// TIA Portal V17 export
// export: Created 2024-08-29T18:23:43.7048748Z, ExportSetting WithDefaults, DisplayName Totally Integrated Automation Portal, DisplayVersion V17 Update 7, DisplayName TIA Portal Openness, DisplayVersion V17 Update 7, DisplayName TIA Portal Version Control Interface, DisplayVersion V17, DisplayName SINAMICS Startdrive Advanced, DisplayVersion V17 SP2, DisplayName SINAMICS Startdrive G110M, G120, G120C, G120D, G120P, G115D, DisplayVersion V17 SP2, DisplayName SINAMICS Startdrive G130, G150, S120, S150, SINAMICS MV, S210, DisplayVersion V17 SP2, DisplayName STEP 7 Professional, DisplayVersion V17 Update 7, DisplayName STEP 7 Safety, DisplayVersion V17 Update 6, DisplayName WinCC Advanced / Unified PC, DisplayVersion V17 Update 7
FUNCTION "analogSignals" : Void   // FC16, LAD
{ S7_Optimized_Access := 'TRUE' }
VERSION : 0.1
// stored: AutoNumber true, IsIECCheckEnabled false, SetENOAutomatically false, UDAEnableTagReadback false
   VAR_TEMP
      minimumScaleRangeArray : Array[0..9] of Real;
      maximumScaleRangeArray : Array[0..9] of Real;
      i : Int;
   END_VAR
BEGIN

REGION Network 1 (SCL): Initialize Temp Values
   FOR #i := 0 TO 9 DO
       #minimumScaleRangeArray[#i] := 0;
       #maximumScaleRangeArray[#i] := 0;
   END_FOR;
END_REGION

REGION Network 2: Load Cell Adquisition
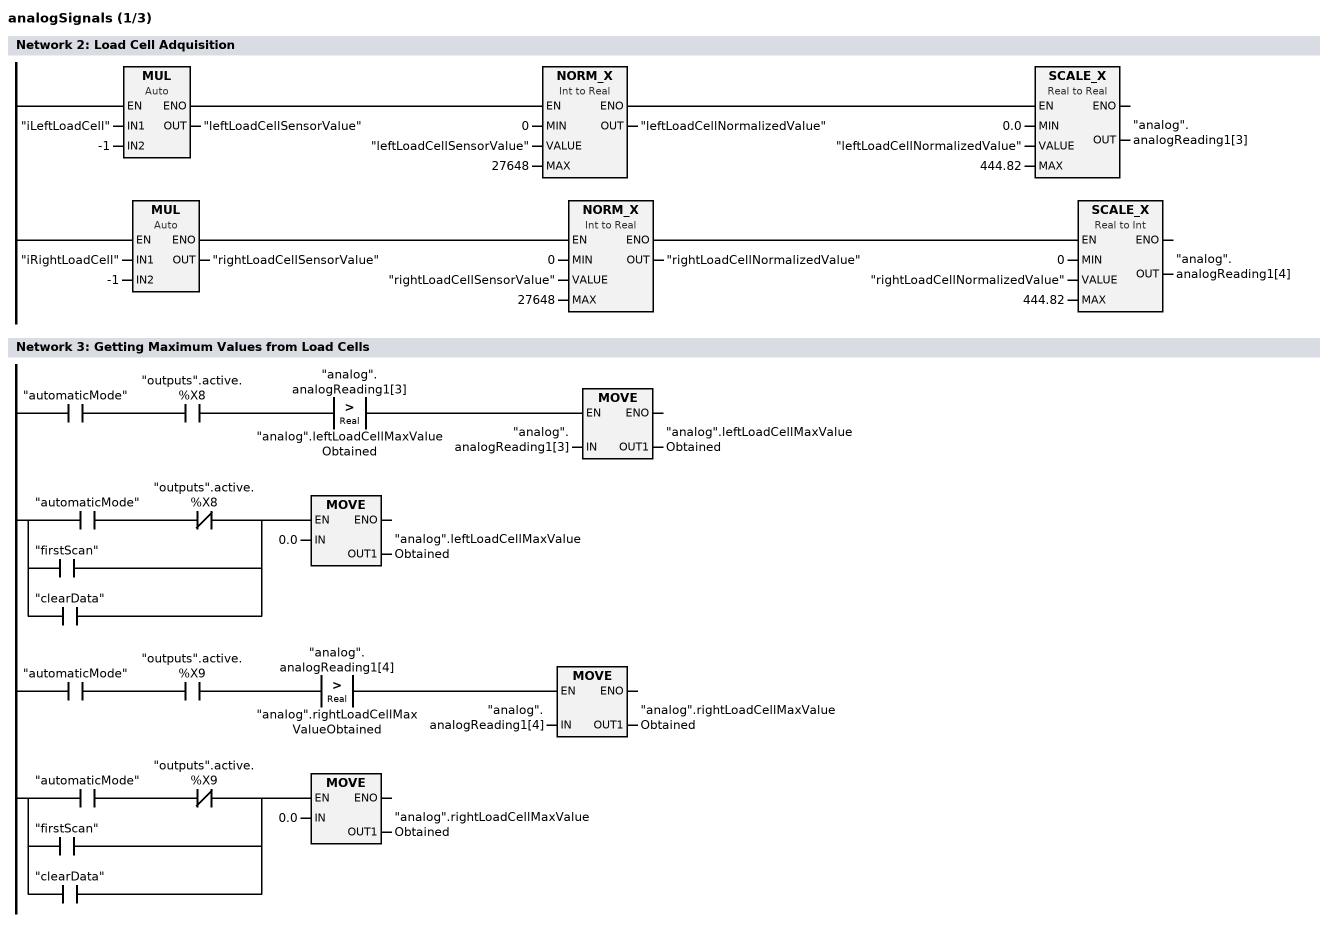
   RUNG wire#powerrail
      Mul(in1 := "iLeftLoadCell", in2 := -1, out => "leftLoadCellSensorValue")
      { S7_Templates := "[SrcType := Int, DestType := Real]" } Normalize(min := 0, value := "leftLoadCellSensorValue", max := 27648, out => "leftLoadCellNormalizedValue")
      { S7_Templates := "[SrcType := Real, DestType := Real]" } Scale(min := 0.0, value := "leftLoadCellNormalizedValue", max := 444.82, out => "analog".analogReading1[3])
   END_RUNG
   RUNG wire#powerrail
      Mul(in1 := "iRightLoadCell", in2 := -1, out => "rightLoadCellSensorValue")
      { S7_Templates := "[SrcType := Int, DestType := Real]" } Normalize(min := 0, value := "rightLoadCellSensorValue", max := 27648, out => "rightLoadCellNormalizedValue")
      { S7_Templates := "[SrcType := Real, DestType := Int]" } Scale(min := 0, value := "rightLoadCellNormalizedValue", max := 444.82, out => "analog".analogReading1[4])
   END_RUNG
   // the same network as SCL:
   "leftLoadCellSensorValue" := "iLeftLoadCell" * (-1);
   "leftLoadCellNormalizedValue" := NORM_X(MIN := 0, VALUE := "leftLoadCellSensorValue", MAX := 27648);
   "analog".analogReading1[3] := SCALE_X(MIN := 0.0, VALUE := "leftLoadCellNormalizedValue", MAX := 444.82);
   "rightLoadCellSensorValue" := "iRightLoadCell" * (-1);
   "rightLoadCellNormalizedValue" := NORM_X(MIN := 0, VALUE := "rightLoadCellSensorValue", MAX := 27648);
   "analog".analogReading1[4] := SCALE_X(MIN := 0, VALUE := "rightLoadCellNormalizedValue", MAX := 444.82);
END_REGION

REGION Network 3: Getting Maximum Values from Load Cells
   RUNG wire#powerrail
      Contact( "automaticMode" )
      Contact( "outputs".active.%X8 )
      { S7_Templates := "SrcType := Real" } GT_Contact(in1 := "analog".analogReading1[3], in2 := "analog".leftLoadCellMaxValueObtained)
      Move(in := "analog".analogReading1[3], out1 => "analog".leftLoadCellMaxValueObtained)
   END_RUNG
   RUNG wire#powerrail
      Contact( "automaticMode" )
      I_Contact( "outputs".active.%X8 )
      wire#w1
      Move(in := 0.0, out1 => "analog".leftLoadCellMaxValueObtained)
   END_RUNG
   RUNG wire#powerrail
      Contact( "firstScan" )
   END_RUNG wire#w1
   RUNG wire#powerrail
      Contact( "clearData" )
   END_RUNG wire#w1
   RUNG wire#powerrail
      Contact( "automaticMode" )
      Contact( "outputs".active.%X9 )
      { S7_Templates := "SrcType := Real" } GT_Contact(in1 := "analog".analogReading1[4], in2 := "analog".rightLoadCellMaxValueObtained)
      Move(in := "analog".analogReading1[4], out1 => "analog".rightLoadCellMaxValueObtained)
   END_RUNG
   RUNG wire#powerrail
      Contact( "automaticMode" )
      I_Contact( "outputs".active.%X9 )
      wire#w2
      Move(in := 0.0, out1 => "analog".rightLoadCellMaxValueObtained)
   END_RUNG
   RUNG wire#powerrail
      Contact( "firstScan" )
   END_RUNG wire#w2
   RUNG wire#powerrail
      Contact( "clearData" )
   END_RUNG wire#w2
   // the same network as SCL:
   IF "automaticMode" AND "outputs".active.%X8 AND ("analog".analogReading1[3] > "analog".leftLoadCellMaxValueObtained) THEN
       "analog".leftLoadCellMaxValueObtained := "analog".analogReading1[3];
   END_IF;
   IF ("automaticMode" AND NOT "outputs".active.%X8) OR "firstScan" OR "clearData" THEN
       "analog".leftLoadCellMaxValueObtained := 0.0;
   END_IF;
   IF "automaticMode" AND "outputs".active.%X9 AND ("analog".analogReading1[4] > "analog".rightLoadCellMaxValueObtained) THEN
       "analog".rightLoadCellMaxValueObtained := "analog".analogReading1[4];
   END_IF;
   IF ("automaticMode" AND NOT "outputs".active.%X9) OR "firstScan" OR "clearData" THEN
       "analog".rightLoadCellMaxValueObtained := 0.0;
   END_IF;
END_REGION

REGION Network 4: Effort OK/NOK Evaluation
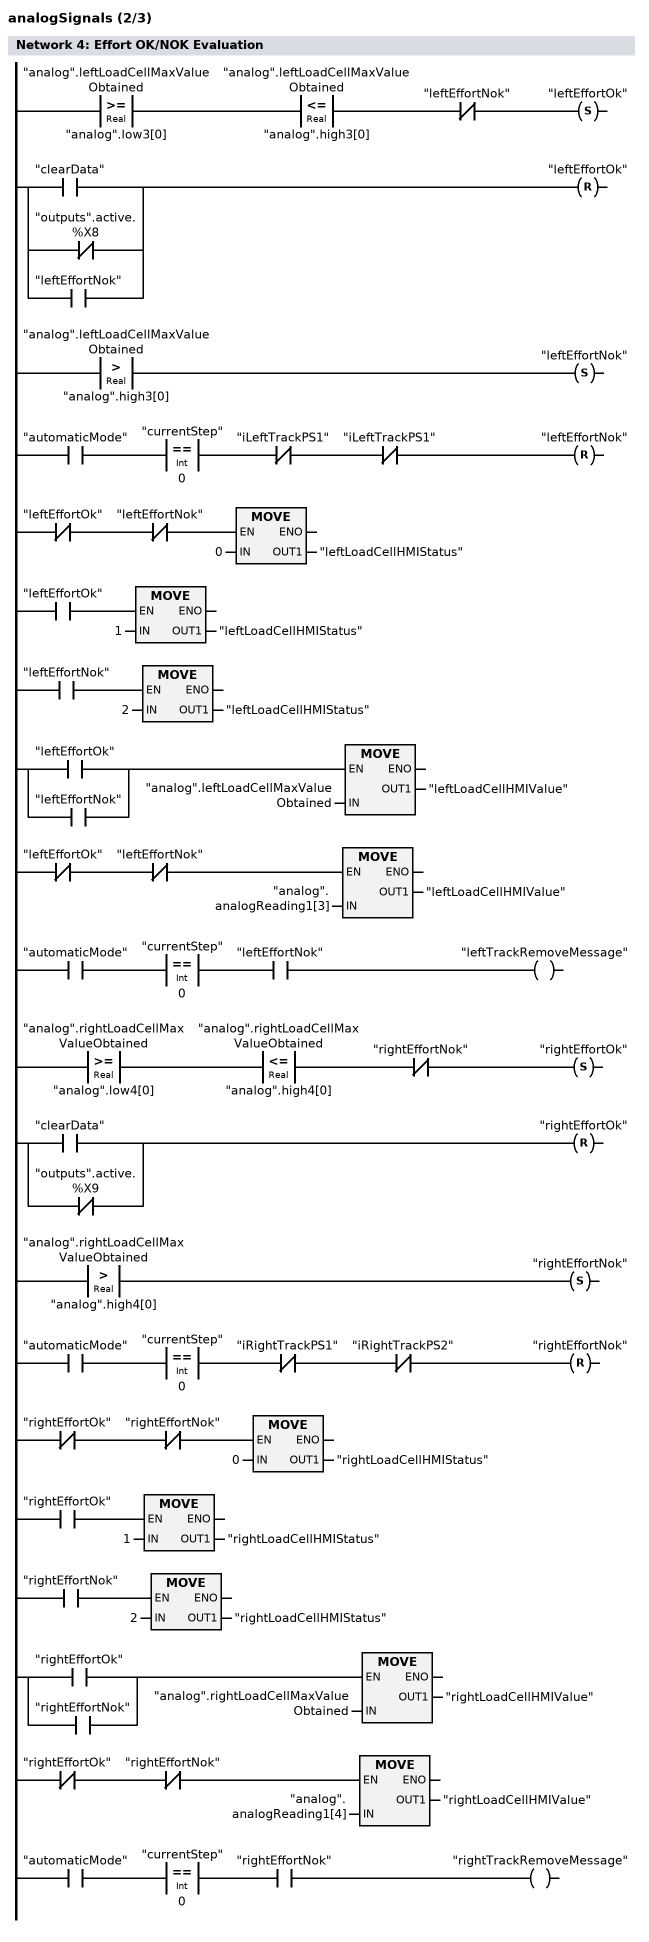
   RUNG wire#powerrail
      { S7_Templates := "SrcType := Real" } GE_Contact(in1 := "analog".leftLoadCellMaxValueObtained, in2 := "analog".low3[0])
      { S7_Templates := "SrcType := Real" } LE_Contact(in1 := "analog".leftLoadCellMaxValueObtained, in2 := "analog".high3[0])
      I_Contact( "leftEffortNok" )
      S_Coil( "leftEffortOk" )
   END_RUNG
   RUNG wire#powerrail
      Contact( "clearData" )
      wire#w1
      R_Coil( "leftEffortOk" )
   END_RUNG
   RUNG wire#powerrail
      I_Contact( "outputs".active.%X8 )
   END_RUNG wire#w1
   RUNG wire#powerrail
      Contact( "leftEffortNok" )
   END_RUNG wire#w1
   RUNG wire#powerrail
      { S7_Templates := "SrcType := Real" } GT_Contact(in1 := "analog".leftLoadCellMaxValueObtained, in2 := "analog".high3[0])
      S_Coil( "leftEffortNok" )
   END_RUNG
   RUNG wire#powerrail
      Contact( "automaticMode" )
      { S7_Templates := "SrcType := Int" } EQ_Contact(in1 := "currentStep", in2 := 0)
      I_Contact( "iLeftTrackPS1" )
      I_Contact( "iLeftTrackPS1" )
      R_Coil( "leftEffortNok" )
   END_RUNG
   RUNG wire#powerrail
      I_Contact( "leftEffortOk" )
      I_Contact( "leftEffortNok" )
      Move(in := 0, out1 => "leftLoadCellHMIStatus")
   END_RUNG
   RUNG wire#powerrail
      Contact( "leftEffortOk" )
      Move(in := 1, out1 => "leftLoadCellHMIStatus")
   END_RUNG
   RUNG wire#powerrail
      Contact( "leftEffortNok" )
      Move(in := 2, out1 => "leftLoadCellHMIStatus")
   END_RUNG
   RUNG wire#powerrail
      Contact( "leftEffortOk" )
      wire#w2
      Move(in := "analog".leftLoadCellMaxValueObtained, out1 => "leftLoadCellHMIValue")
   END_RUNG
   RUNG wire#powerrail
      Contact( "leftEffortNok" )
   END_RUNG wire#w2
   RUNG wire#powerrail
      I_Contact( "leftEffortOk" )
      I_Contact( "leftEffortNok" )
      Move(in := "analog".analogReading1[3], out1 => "leftLoadCellHMIValue")
   END_RUNG
   RUNG wire#powerrail
      Contact( "automaticMode" )
      { S7_Templates := "SrcType := Int" } EQ_Contact(in1 := "currentStep", in2 := 0)
      Contact( "leftEffortNok" )
      Coil( "leftTrackRemoveMessage" )
   END_RUNG
   RUNG wire#powerrail
      { S7_Templates := "SrcType := Real" } GE_Contact(in1 := "analog".rightLoadCellMaxValueObtained, in2 := "analog".low4[0])
      { S7_Templates := "SrcType := Real" } LE_Contact(in1 := "analog".rightLoadCellMaxValueObtained, in2 := "analog".high4[0])
      I_Contact( "rightEffortNok" )
      S_Coil( "rightEffortOk" )
   END_RUNG
   RUNG wire#powerrail
      Contact( "clearData" )
      wire#w3
      R_Coil( "rightEffortOk" )
   END_RUNG
   RUNG wire#powerrail
      I_Contact( "outputs".active.%X9 )
   END_RUNG wire#w3
   RUNG wire#powerrail
      { S7_Templates := "SrcType := Real" } GT_Contact(in1 := "analog".rightLoadCellMaxValueObtained, in2 := "analog".high4[0])
      S_Coil( "rightEffortNok" )
   END_RUNG
   RUNG wire#powerrail
      Contact( "automaticMode" )
      { S7_Templates := "SrcType := Int" } EQ_Contact(in1 := "currentStep", in2 := 0)
      I_Contact( "iRightTrackPS1" )
      I_Contact( "iRightTrackPS2" )
      R_Coil( "rightEffortNok" )
   END_RUNG
   RUNG wire#powerrail
      I_Contact( "rightEffortOk" )
      I_Contact( "rightEffortNok" )
      Move(in := 0, out1 => "rightLoadCellHMIStatus")
   END_RUNG
   RUNG wire#powerrail
      Contact( "rightEffortOk" )
      Move(in := 1, out1 => "rightLoadCellHMIStatus")
   END_RUNG
   RUNG wire#powerrail
      Contact( "rightEffortNok" )
      Move(in := 2, out1 => "rightLoadCellHMIStatus")
   END_RUNG
   RUNG wire#powerrail
      Contact( "rightEffortOk" )
      wire#w4
      Move(in := "analog".rightLoadCellMaxValueObtained, out1 => "rightLoadCellHMIValue")
   END_RUNG
   RUNG wire#powerrail
      Contact( "rightEffortNok" )
   END_RUNG wire#w4
   RUNG wire#powerrail
      I_Contact( "rightEffortOk" )
      I_Contact( "rightEffortNok" )
      Move(in := "analog".analogReading1[4], out1 => "rightLoadCellHMIValue")
   END_RUNG
   RUNG wire#powerrail
      Contact( "automaticMode" )
      { S7_Templates := "SrcType := Int" } EQ_Contact(in1 := "currentStep", in2 := 0)
      Contact( "rightEffortNok" )
      Coil( "rightTrackRemoveMessage" )
   END_RUNG
   // the same network as SCL:
   IF ("analog".leftLoadCellMaxValueObtained >= "analog".low3[0]) AND ("analog".leftLoadCellMaxValueObtained <= "analog".high3[0]) AND NOT "leftEffortNok" THEN
       "leftEffortOk" := TRUE;
   END_IF;
   IF "clearData" OR NOT "outputs".active.%X8 OR "leftEffortNok" THEN "leftEffortOk" := FALSE; END_IF;
   IF "analog".leftLoadCellMaxValueObtained > "analog".high3[0] THEN "leftEffortNok" := TRUE; END_IF;
   IF "automaticMode" AND ("currentStep" = 0) AND NOT "iLeftTrackPS1" AND NOT "iLeftTrackPS1" THEN
       "leftEffortNok" := FALSE;
   END_IF;
   IF NOT "leftEffortOk" AND NOT "leftEffortNok" THEN "leftLoadCellHMIStatus" := 0; END_IF;
   IF "leftEffortOk" THEN "leftLoadCellHMIStatus" := 1; END_IF;
   IF "leftEffortNok" THEN "leftLoadCellHMIStatus" := 2; END_IF;
   IF "leftEffortOk" OR "leftEffortNok" THEN
       "leftLoadCellHMIValue" := "analog".leftLoadCellMaxValueObtained;
   END_IF;
   IF NOT "leftEffortOk" AND NOT "leftEffortNok" THEN
       "leftLoadCellHMIValue" := "analog".analogReading1[3];
   END_IF;
   "leftTrackRemoveMessage" := "automaticMode" AND ("currentStep" = 0) AND "leftEffortNok";
   IF ("analog".rightLoadCellMaxValueObtained >= "analog".low4[0]) AND ("analog".rightLoadCellMaxValueObtained <= "analog".high4[0]) AND NOT "rightEffortNok" THEN
       "rightEffortOk" := TRUE;
   END_IF;
   IF "clearData" OR NOT "outputs".active.%X9 THEN "rightEffortOk" := FALSE; END_IF;
   IF "analog".rightLoadCellMaxValueObtained > "analog".high4[0] THEN "rightEffortNok" := TRUE; END_IF;
   IF "automaticMode" AND ("currentStep" = 0) AND NOT "iRightTrackPS1" AND NOT "iRightTrackPS2" THEN
       "rightEffortNok" := FALSE;
   END_IF;
   IF NOT "rightEffortOk" AND NOT "rightEffortNok" THEN "rightLoadCellHMIStatus" := 0; END_IF;
   IF "rightEffortOk" THEN "rightLoadCellHMIStatus" := 1; END_IF;
   IF "rightEffortNok" THEN "rightLoadCellHMIStatus" := 2; END_IF;
   IF "rightEffortOk" OR "rightEffortNok" THEN
       "rightLoadCellHMIValue" := "analog".rightLoadCellMaxValueObtained;
   END_IF;
   IF NOT "rightEffortOk" AND NOT "rightEffortNok" THEN
       "rightLoadCellHMIValue" := "analog".analogReading1[4];
   END_IF;
   "rightTrackRemoveMessage" := "automaticMode" AND ("currentStep" = 0) AND "rightEffortNok";
END_REGION

REGION Network 5: SENSOR DISTANCES
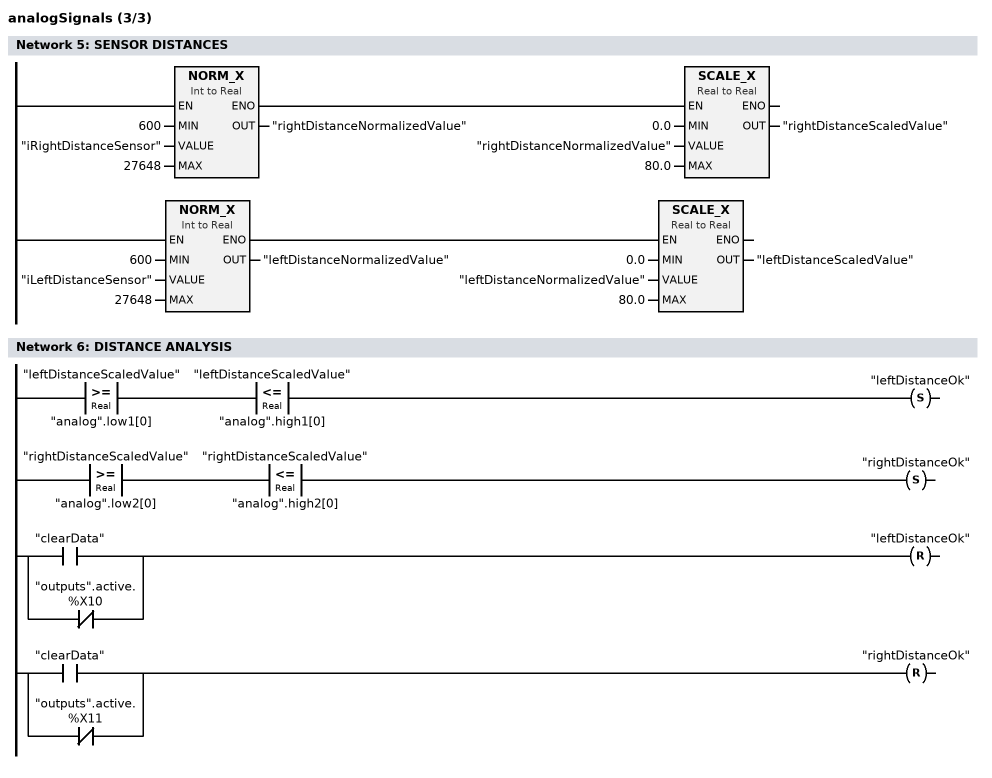
   RUNG wire#powerrail
      { S7_Templates := "[SrcType := Int, DestType := Real]" } Normalize(min := 600, value := "iRightDistanceSensor", max := 27648, out => "rightDistanceNormalizedValue")
      { S7_Templates := "[SrcType := Real, DestType := Real]" } Scale(min := 0.0, value := "rightDistanceNormalizedValue", max := 80.0, out => "rightDistanceScaledValue")
   END_RUNG
   RUNG wire#powerrail
      { S7_Templates := "[SrcType := Int, DestType := Real]" } Normalize(min := 600, value := "iLeftDistanceSensor", max := 27648, out => "leftDistanceNormalizedValue")
      { S7_Templates := "[SrcType := Real, DestType := Real]" } Scale(min := 0.0, value := "leftDistanceNormalizedValue", max := 80.0, out => "leftDistanceScaledValue")
   END_RUNG
   // the same network as SCL:
   "rightDistanceNormalizedValue" := NORM_X(MIN := 600, VALUE := "iRightDistanceSensor", MAX := 27648);
   "rightDistanceScaledValue" := SCALE_X(MIN := 0.0, VALUE := "rightDistanceNormalizedValue", MAX := 80.0);
   "leftDistanceNormalizedValue" := NORM_X(MIN := 600, VALUE := "iLeftDistanceSensor", MAX := 27648);
   "leftDistanceScaledValue" := SCALE_X(MIN := 0.0, VALUE := "leftDistanceNormalizedValue", MAX := 80.0);
END_REGION

REGION Network 6: DISTANCE ANALYSIS
   RUNG wire#powerrail
      { S7_Templates := "SrcType := Real" } GE_Contact(in1 := "leftDistanceScaledValue", in2 := "analog".low1[0])
      { S7_Templates := "SrcType := Real" } LE_Contact(in1 := "leftDistanceScaledValue", in2 := "analog".high1[0])
      S_Coil( "leftDistanceOk" )
   END_RUNG
   RUNG wire#powerrail
      { S7_Templates := "SrcType := Real" } GE_Contact(in1 := "rightDistanceScaledValue", in2 := "analog".low2[0])
      { S7_Templates := "SrcType := Real" } LE_Contact(in1 := "rightDistanceScaledValue", in2 := "analog".high2[0])
      S_Coil( "rightDistanceOk" )
   END_RUNG
   RUNG wire#powerrail
      Contact( "clearData" )
      wire#w1
      R_Coil( "leftDistanceOk" )
   END_RUNG
   RUNG wire#powerrail
      I_Contact( "outputs".active.%X10 )
   END_RUNG wire#w1
   RUNG wire#powerrail
      Contact( "clearData" )
      wire#w2
      R_Coil( "rightDistanceOk" )
   END_RUNG
   RUNG wire#powerrail
      I_Contact( "outputs".active.%X11 )
   END_RUNG wire#w2
   // the same network as SCL:
   IF ("leftDistanceScaledValue" >= "analog".low1[0]) AND ("leftDistanceScaledValue" <= "analog".high1[0]) THEN
       "leftDistanceOk" := TRUE;
   END_IF;
   IF ("rightDistanceScaledValue" >= "analog".low2[0]) AND ("rightDistanceScaledValue" <= "analog".high2[0]) THEN
       "rightDistanceOk" := TRUE;
   END_IF;
   IF "clearData" OR NOT "outputs".active.%X10 THEN "leftDistanceOk" := FALSE; END_IF;
   IF "clearData" OR NOT "outputs".active.%X11 THEN "rightDistanceOk" := FALSE; END_IF;
END_REGION
END_FUNCTION
